(* Logix 5000 project; controller RN21_Architecture 1769-L16ER-BB1B rev 35.11; software revision 35.00; part 7 of 9 *)
(* tags used below, declared in another part *)
   ALMSrc_UniqueNum : DINT;
   AUDSrc : UDT_Audit;
   AUDSrc_UniqueNum : DINT;
   BMANSrc : UDT_Batch;
   BMANSrc_UniqueNum : DINT;
   FC_BMAN_Arch : AOI_BMAN_Arch;
   FC_TBC : AOI_TBC;
   FCI_AUDDataLogTrig : BOOL;
   FCI_BMANDataLogTrig : BOOL;
   HMI_CONTROL_SCREEN : DINT;
   HmiCurrentScreen : DINT;
   HMIOLDSCREENVALUE : DINT;
   HMISCREEN : BOOL;
   HMISCREENCHANGED : BOOL;
   inactivity_in_minutes : DINT;
   inactivity_time : DINT;
   INTERNAL_RN21_HB_PLC2ServerCommFailed : BOOL;
   INTERNAL_RN21_PLC2HMICommFailed : BOOL;
   LBSrc_UniqueNum : DINT;
   LoginDNDel : TIMER;
   PDLSrc_PDL_UID : DINT;
   PLC_HMI_CommTag : BOOL;
   PLC_RTC : DINT[7];
   Remaining_time : DINT;
   remaining_time_compareTag : DINT;
   RN21_AUD_BAMTrig : DINT[5];
   RN21_AUD_BAT_NTrig : DINT[4];
   RN21_AUD_BAT_PTrig : DINT[4];
   RN21_AUD_NETrig : DINT[11];
   RN21_AUDBAM_ONS : BOOL[128];
   RN21_AutoLogedOut : BOOL;
   RN21_BACK_BatchDataStatus : BOOL;   // BATCH START ACKNOWLEDGEMENT STATUS FROM SERVER
   RN21_BACK_BatchStartHMI : BOOL;   // HMI BATCH START IN BATCH DETAILS
   RN21_BACKONS : DINT[1];
   RN21_BMAN_BatchStarted : BOOL;   // BATCH STARTED IN BATCH MANAGEMENT
   RN21_BMAN_BatchStopped : BOOL;   // BATCH STOPPED IN BATCH MANAGEMENT
   RN21_BMAN_HMIBatchStart : BOOL;   // BATCH START
   RN21_BMAN_HMIBatchStop : BOOL;
   RN21_BMANBASTPNEG : BOOL;
   RN21_BMANBASTPPOS : BOOL;
   RN21_BMANBASTRTNEG : BOOL;
   RN21_BMANBASTRTPOS : BOOL;
   RN21_HB_PLC2ServerCommFailed : BOOL;
   RN21_LBStatus : INT;   // Login Block Status
   RN21_Map_BAM : BOOL[128];
   RN21_PLC2HMICommFailed : BOOL;
   RN21_RM_HMICODE : STRING;
   RN21_UMLogoutTag : INT;
   RPSrc_RP_UID : DINT;
   RTC_DATE_AND_TIME_UNLATCH_DELAY1 : TIMER;
   TMR_AutoLogout : TIMER;
   TMR_AutoLogoutRstDly : TIMER;
   TMR_BatchStartAckDlyRst : TIMER;
   TMR_BatchStrtdDlyStsMov : TIMER;
   TMR_HBSetDelay : TIMER;
   TMR_LogoutTagRst : TIMER;
   TMR_PHSetDelay : TIMER;
   TMR_PLCtoHMICommCheck : TIMER;
   TMR_PLCToSrvComCheck : TIMER;
   ALM_TriggerId : BOOL;
   ALM_UniqueNum : DINT;
   AUD_TriggerId : BOOL;
   AUD_UniqueNum : DINT;
   BACK_BATCH_NO : STRING;
   BACK_BatchStartACK : DINT;
   BACK_LOT_NO : STRING;
   BMAN_BatchUniqueId : DINT;
   BMAN_TriggerBit : BOOL;
   BMANSer : UDT_Batch;
   HB_HEART_BEAT : BOOL;
   LOGIN_TriggerId : BOOL;
   LOGIN_UniqueNum : DINT;
   PDL_Trigger : BOOL;
   PDL_UID : DINT;
   RN21_BACK_BatchSize : REAL;
   RN21_BACK_ProductCode : STRING;
   RN21_BACK_ProductName : STRING;
   RP_Trigger : BOOL;
   RP_UID : DINT;
   RTC_DAY : DINT;
   RTC_HOUR : DINT;
   RTC_MINUTE : DINT;
   RTC_MONTH : DINT;
   RTC_SAVE_DATE_AND_TIME : BOOL;
   RTC_SECONDS : DINT;
   RTC_UniqueId : DINT;
   RTC_YEAR : DINT;
   ServerRTC : DINT[8];
   TBC_ALARMBLOCK_PLCUID : DINT;
   TBC_ALARMBLOCK_SERVERUID : DINT;
   TBC_ALARMBLOCK_TRIGGER : BOOL;
   TBC_AUDITBLOCK_PLCUID : DINT;
   TBC_AUDITBLOCK_SERVERUID : DINT;
   TBC_AUDITBLOCK_TRIGGER : BOOL;
   TBC_BATCHMGMTBLOCK_PLCUID : DINT;
   TBC_BATCHMGMTBLOCK_SERVERUID : DINT;
   TBC_BATCHMGMTBLOCK_TRIGGER : BOOL;
   TBC_POSITION : DINT;
   TBC_PROCESSBLOCK_PLCUID : DINT;
   TBC_PROCESSBLOCK_SERVERUID : DINT;
   TBC_PROCESSBLOCK_TRIGGER : BOOL;
   TBC_RECIPEBLOCK_PLCUID : DINT;
   TBC_RECIPEBLOCK_SERVERUID : DINT;
   TBC_RECIPEBLOCK_TRIGGER : BOOL;
   TBC_UID : DINT;
   TBC_UMBLOCK_PLCUID : DINT;
   TBC_UMBLOCK_SERVERUID : DINT;
   TBC_UMBLOCK_TRIGGER : BOOL;
(* MainProgram, continued *)

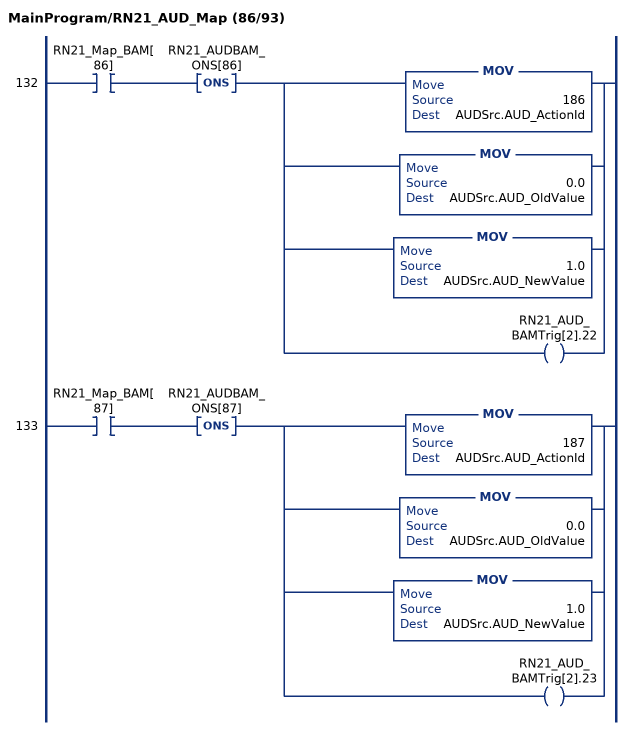
   [picture p168: MainProgram/RN21_AUD_Map rungs 132-133]
   132: XIC(RN21_Map_BAM[86])ONS(RN21_AUDBAM_ONS[86])[MOV(186,AUDSrc.AUD_ActionId) ,MOV(0.0,AUDSrc.AUD_OldValue) ,MOV(1.0,AUDSrc.AUD_NewValue) ,OTE(RN21_AUD_BAMTrig[2].22) ];
   133: XIC(RN21_Map_BAM[87])ONS(RN21_AUDBAM_ONS[87])[MOV(187,AUDSrc.AUD_ActionId) ,MOV(0.0,AUDSrc.AUD_OldValue) ,MOV(1.0,AUDSrc.AUD_NewValue) ,OTE(RN21_AUD_BAMTrig[2].23) ];
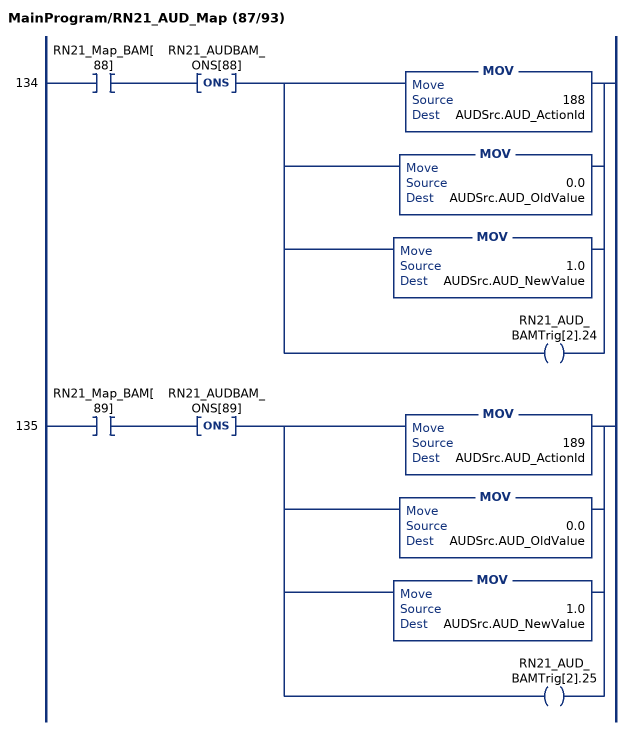
   134: XIC(RN21_Map_BAM[88])ONS(RN21_AUDBAM_ONS[88])[MOV(188,AUDSrc.AUD_ActionId) ,MOV(0.0,AUDSrc.AUD_OldValue) ,MOV(1.0,AUDSrc.AUD_NewValue) ,OTE(RN21_AUD_BAMTrig[2].24) ];
   135: XIC(RN21_Map_BAM[89])ONS(RN21_AUDBAM_ONS[89])[MOV(189,AUDSrc.AUD_ActionId) ,MOV(0.0,AUDSrc.AUD_OldValue) ,MOV(1.0,AUDSrc.AUD_NewValue) ,OTE(RN21_AUD_BAMTrig[2].25) ];
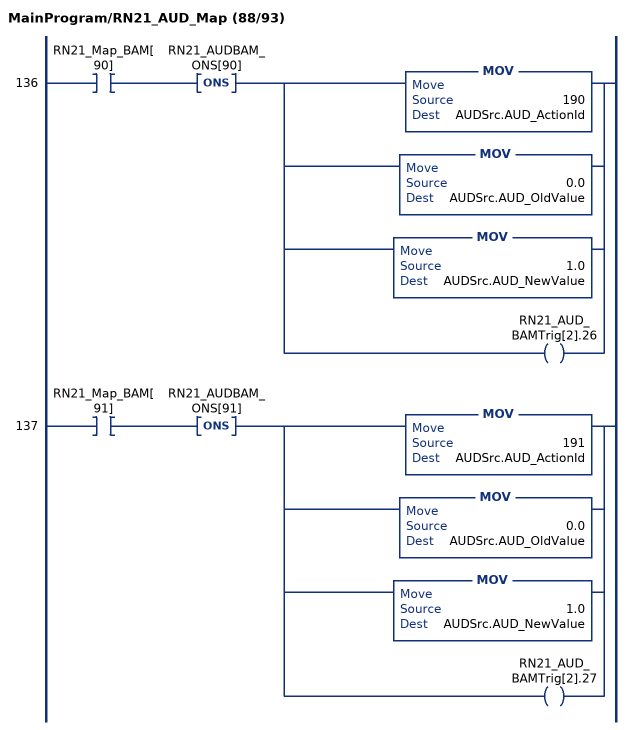
   136: XIC(RN21_Map_BAM[90])ONS(RN21_AUDBAM_ONS[90])[MOV(190,AUDSrc.AUD_ActionId) ,MOV(0.0,AUDSrc.AUD_OldValue) ,MOV(1.0,AUDSrc.AUD_NewValue) ,OTE(RN21_AUD_BAMTrig[2].26) ];
   137: XIC(RN21_Map_BAM[91])ONS(RN21_AUDBAM_ONS[91])[MOV(191,AUDSrc.AUD_ActionId) ,MOV(0.0,AUDSrc.AUD_OldValue) ,MOV(1.0,AUDSrc.AUD_NewValue) ,OTE(RN21_AUD_BAMTrig[2].27) ];
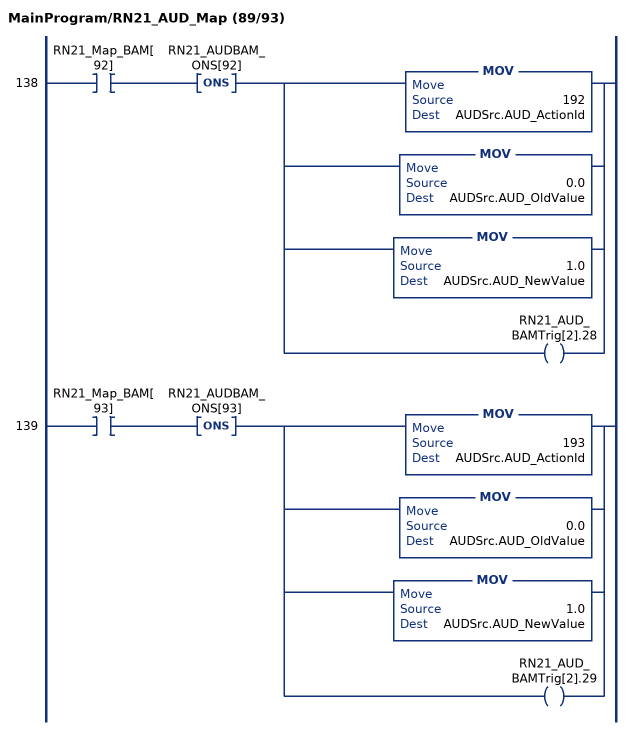
   138: XIC(RN21_Map_BAM[92])ONS(RN21_AUDBAM_ONS[92])[MOV(192,AUDSrc.AUD_ActionId) ,MOV(0.0,AUDSrc.AUD_OldValue) ,MOV(1.0,AUDSrc.AUD_NewValue) ,OTE(RN21_AUD_BAMTrig[2].28) ];
   139: XIC(RN21_Map_BAM[93])ONS(RN21_AUDBAM_ONS[93])[MOV(193,AUDSrc.AUD_ActionId) ,MOV(0.0,AUDSrc.AUD_OldValue) ,MOV(1.0,AUDSrc.AUD_NewValue) ,OTE(RN21_AUD_BAMTrig[2].29) ];
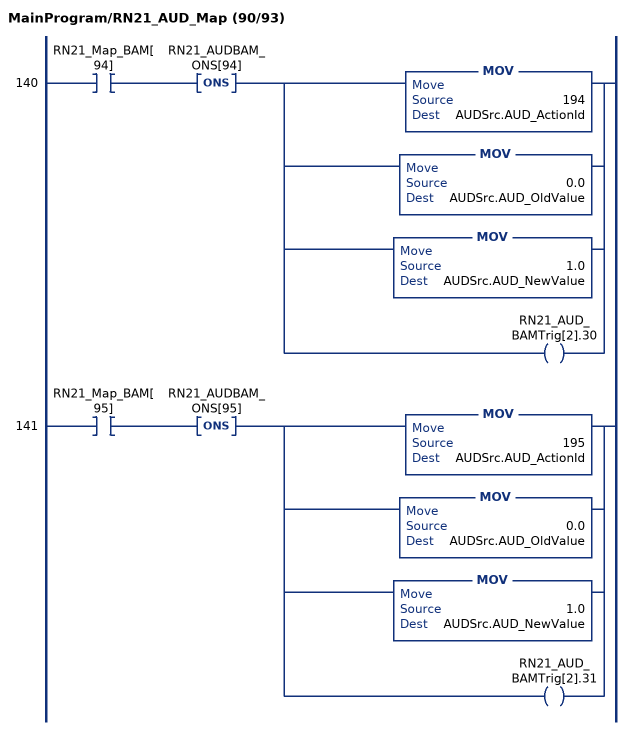
   140: XIC(RN21_Map_BAM[94])ONS(RN21_AUDBAM_ONS[94])[MOV(194,AUDSrc.AUD_ActionId) ,MOV(0.0,AUDSrc.AUD_OldValue) ,MOV(1.0,AUDSrc.AUD_NewValue) ,OTE(RN21_AUD_BAMTrig[2].30) ];
   141: XIC(RN21_Map_BAM[95])ONS(RN21_AUDBAM_ONS[95])[MOV(195,AUDSrc.AUD_ActionId) ,MOV(0.0,AUDSrc.AUD_OldValue) ,MOV(1.0,AUDSrc.AUD_NewValue) ,OTE(RN21_AUD_BAMTrig[2].31) ];
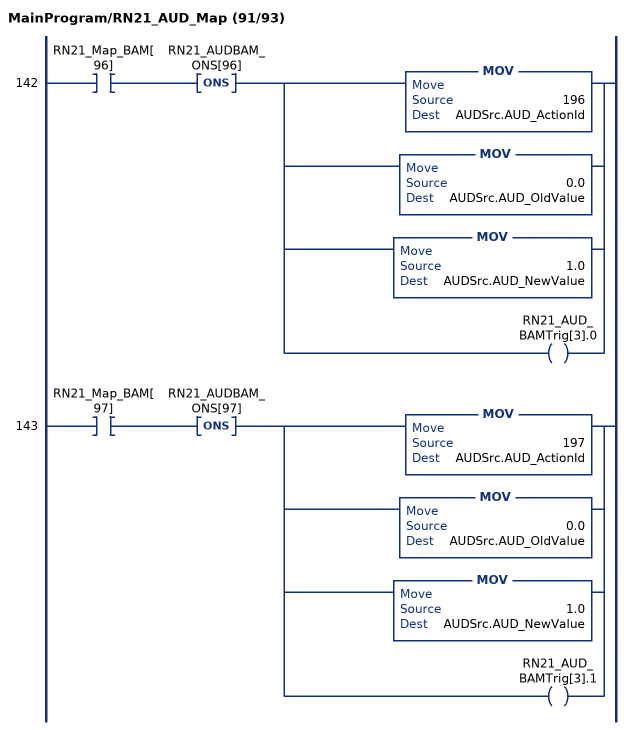
   142: XIC(RN21_Map_BAM[96])ONS(RN21_AUDBAM_ONS[96])[MOV(196,AUDSrc.AUD_ActionId) ,MOV(0.0,AUDSrc.AUD_OldValue) ,MOV(1.0,AUDSrc.AUD_NewValue) ,OTE(RN21_AUD_BAMTrig[3].0) ];
   143: XIC(RN21_Map_BAM[97])ONS(RN21_AUDBAM_ONS[97])[MOV(197,AUDSrc.AUD_ActionId) ,MOV(0.0,AUDSrc.AUD_OldValue) ,MOV(1.0,AUDSrc.AUD_NewValue) ,OTE(RN21_AUD_BAMTrig[3].1) ];
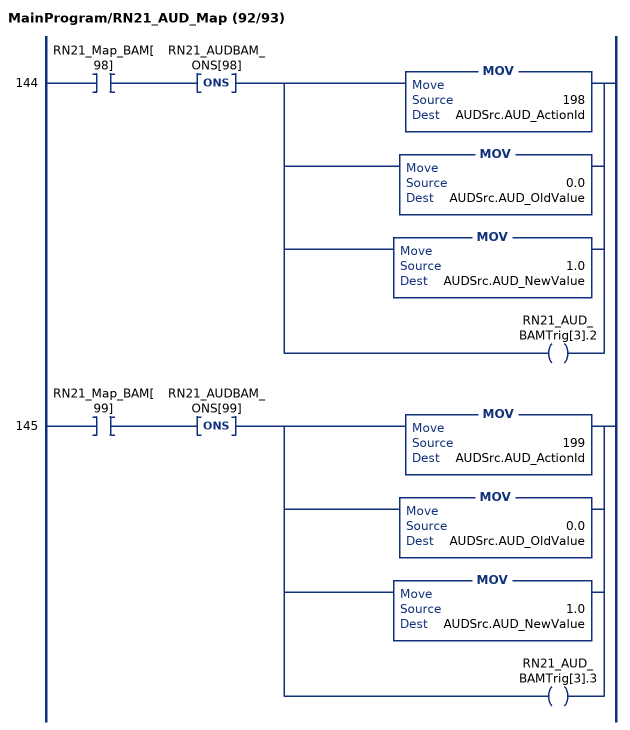
   144: XIC(RN21_Map_BAM[98])ONS(RN21_AUDBAM_ONS[98])[MOV(198,AUDSrc.AUD_ActionId) ,MOV(0.0,AUDSrc.AUD_OldValue) ,MOV(1.0,AUDSrc.AUD_NewValue) ,OTE(RN21_AUD_BAMTrig[3].2) ];
   145: XIC(RN21_Map_BAM[99])ONS(RN21_AUDBAM_ONS[99])[MOV(199,AUDSrc.AUD_ActionId) ,MOV(0.0,AUDSrc.AUD_OldValue) ,MOV(1.0,AUDSrc.AUD_NewValue) ,OTE(RN21_AUD_BAMTrig[3].3) ];
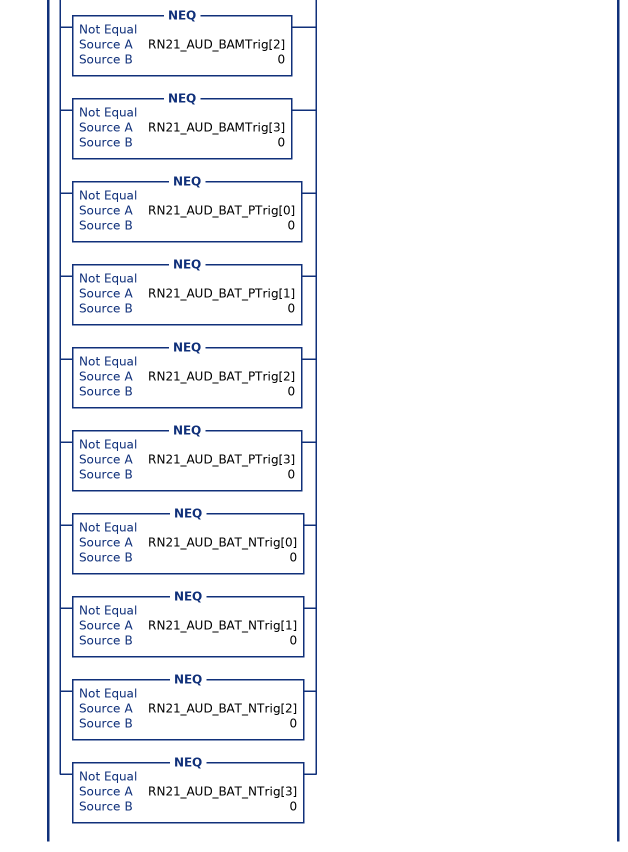
   146: [NEQ(RN21_AUD_NETrig[0],0) ,NEQ(RN21_AUD_NETrig[1],0) ,NEQ(RN21_AUD_NETrig[2],0) ,NEQ(RN21_AUD_NETrig[3],0) ,NEQ(RN21_AUD_NETrig[4],0) ,NEQ(RN21_AUD_NETrig[5],0) ,NEQ(RN21_AUD_NETrig[6],0) ,NEQ(RN21_AUD_NETrig[7],0) ,NEQ(RN21_AUD_NETrig[8],0) ,NEQ(RN21_AUD_NETrig[9],0) ,NEQ(RN21_AUD_BAMTrig[0],0) ,NEQ(RN21_AUD_BAMTrig[1],0) ,NEQ(RN21_AUD_BAMTrig[2],0) ,NEQ(RN21_AUD_BAMTrig[3],0) ,NEQ(RN21_AUD_BAT_PTrig[0],0) ,NEQ(RN21_AUD_BAT_PTrig[1],0) ,NEQ(RN21_AUD_BAT_PTrig[2],0) ,NEQ(RN21_AUD_BAT_PTrig[3],0) ,NEQ(RN21_AUD_BAT_NTrig[0],0) ,NEQ(RN21_AUD_BAT_NTrig[1],0) ,NEQ(RN21_AUD_BAT_NTrig[2],0) ,NEQ(RN21_AUD_BAT_NTrig[3],0) ]OTE(FCI_AUDDataLogTrig);
END_ROUTINE

ROUTINE RN21_BMAN_Main   (* ladder *)
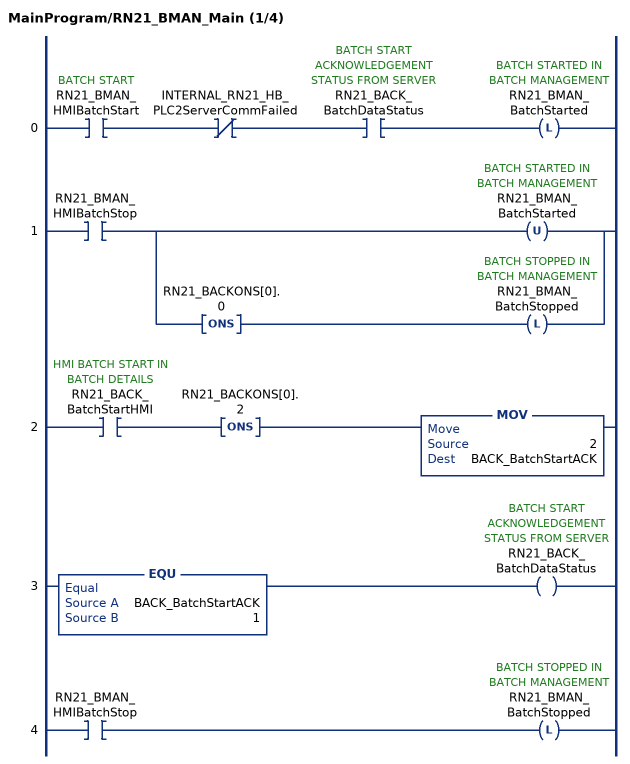
   0: XIC(RN21_BMAN_HMIBatchStart)XIO(INTERNAL_RN21_HB_PLC2ServerCommFailed)XIC(RN21_BACK_BatchDataStatus)OTL(RN21_BMAN_BatchStarted);
   1: XIC(RN21_BMAN_HMIBatchStop)[OTU(RN21_BMAN_BatchStarted) ,ONS(RN21_BACKONS[0].0) OTL(RN21_BMAN_BatchStopped) ];
   2: XIC(RN21_BACK_BatchStartHMI)ONS(RN21_BACKONS[0].2)MOV(2,BACK_BatchStartACK);
   3: EQU(BACK_BatchStartACK,1)OTE(RN21_BACK_BatchDataStatus);
   4: XIC(RN21_BMAN_HMIBatchStop)OTL(RN21_BMAN_BatchStopped);
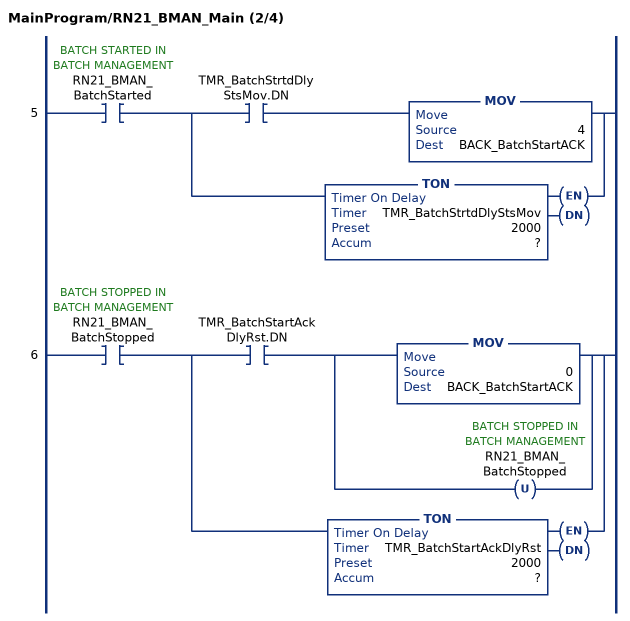
   5: XIC(RN21_BMAN_BatchStarted)[XIC(TMR_BatchStrtdDlyStsMov.DN) MOV(4,BACK_BatchStartACK) ,TON(TMR_BatchStrtdDlyStsMov,?,?) ];
   6: XIC(RN21_BMAN_BatchStopped)[XIC(TMR_BatchStartAckDlyRst.DN) [MOV(0,BACK_BatchStartACK) ,OTU(RN21_BMAN_BatchStopped) ] ,TON(TMR_BatchStartAckDlyRst,?,?) ];
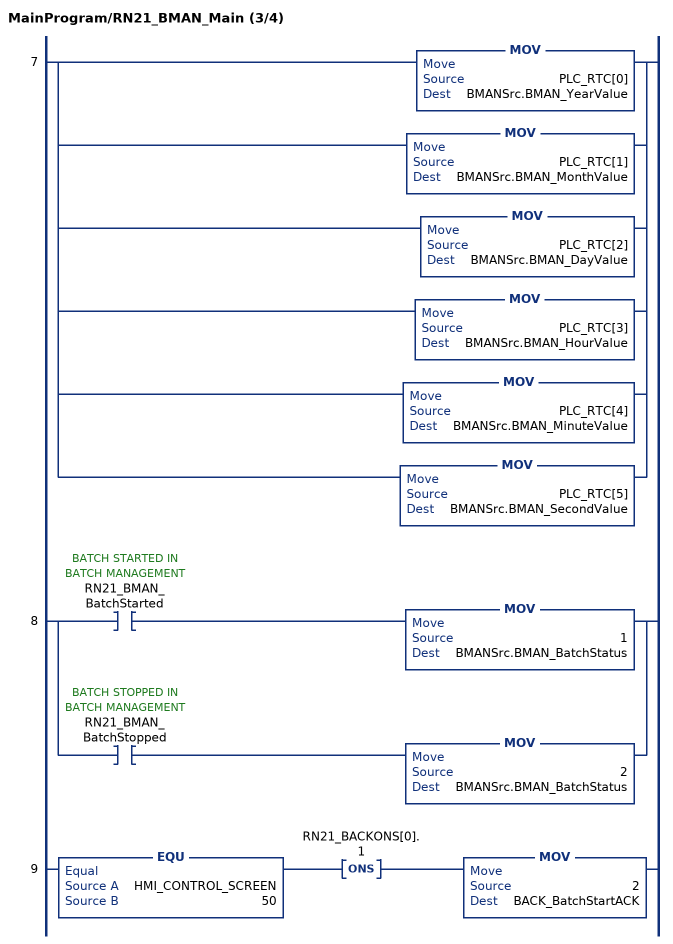
   7: [MOV(PLC_RTC[0],BMANSrc.BMAN_YearValue) ,MOV(PLC_RTC[1],BMANSrc.BMAN_MonthValue) ,MOV(PLC_RTC[2],BMANSrc.BMAN_DayValue) ,MOV(PLC_RTC[3],BMANSrc.BMAN_HourValue) ,MOV(PLC_RTC[4],BMANSrc.BMAN_MinuteValue) ,MOV(PLC_RTC[5],BMANSrc.BMAN_SecondValue) ];
   8: [XIC(RN21_BMAN_BatchStarted) MOV(1,BMANSrc.BMAN_BatchStatus) ,XIC(RN21_BMAN_BatchStopped) MOV(2,BMANSrc.BMAN_BatchStatus) ];
   9: EQU(HMI_CONTROL_SCREEN,50)ONS(RN21_BACKONS[0].1)MOV(2,BACK_BatchStartACK);
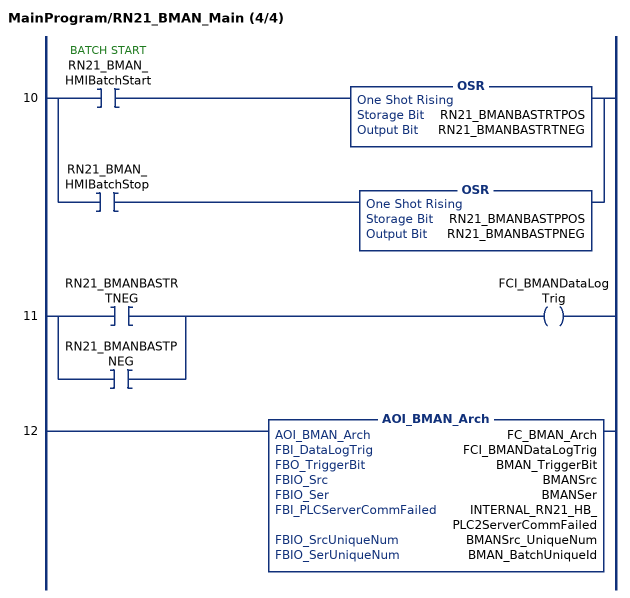
   10: [XIC(RN21_BMAN_HMIBatchStart) OSR(RN21_BMANBASTRTPOS,RN21_BMANBASTRTNEG) ,XIC(RN21_BMAN_HMIBatchStop) OSR(RN21_BMANBASTPPOS,RN21_BMANBASTPNEG) ];
   11: [XIC(RN21_BMANBASTRTNEG) ,XIC(RN21_BMANBASTPNEG) ]OTE(FCI_BMANDataLogTrig);
   12: AOI_BMAN_Arch(FC_BMAN_Arch,FCI_BMANDataLogTrig,BMAN_TriggerBit,BMANSrc,BMANSer,INTERNAL_RN21_HB_PLC2ServerCommFailed,BMANSrc_UniqueNum,BMAN_BatchUniqueId);
END_ROUTINE

ROUTINE RN21_BMAN_Map   (* ladder *)
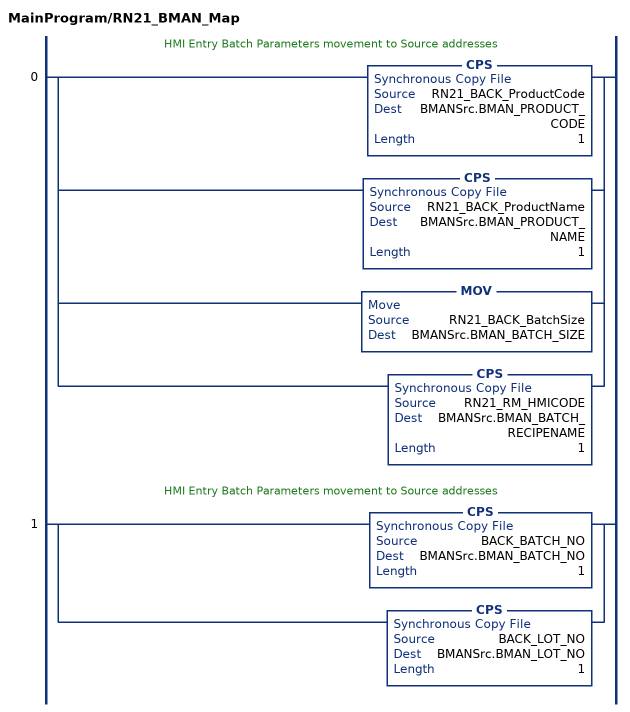
   // HMI Entry Batch Parameters movement to Source addresses
   0: [CPS(RN21_BACK_ProductCode,BMANSrc.BMAN_PRODUCT_CODE,1) ,CPS(RN21_BACK_ProductName,BMANSrc.BMAN_PRODUCT_NAME,1) ,MOV(RN21_BACK_BatchSize,BMANSrc.BMAN_BATCH_SIZE) ,CPS(RN21_RM_HMICODE,BMANSrc.BMAN_BATCH_RECIPENAME,1) ];
   // HMI Entry Batch Parameters movement to Source addresses
   1: [CPS(BACK_BATCH_NO,BMANSrc.BMAN_BATCH_NO,1) ,CPS(BACK_LOT_NO,BMANSrc.BMAN_LOT_NO,1) ];
END_ROUTINE

ROUTINE RN21_Global   (* ladder *)
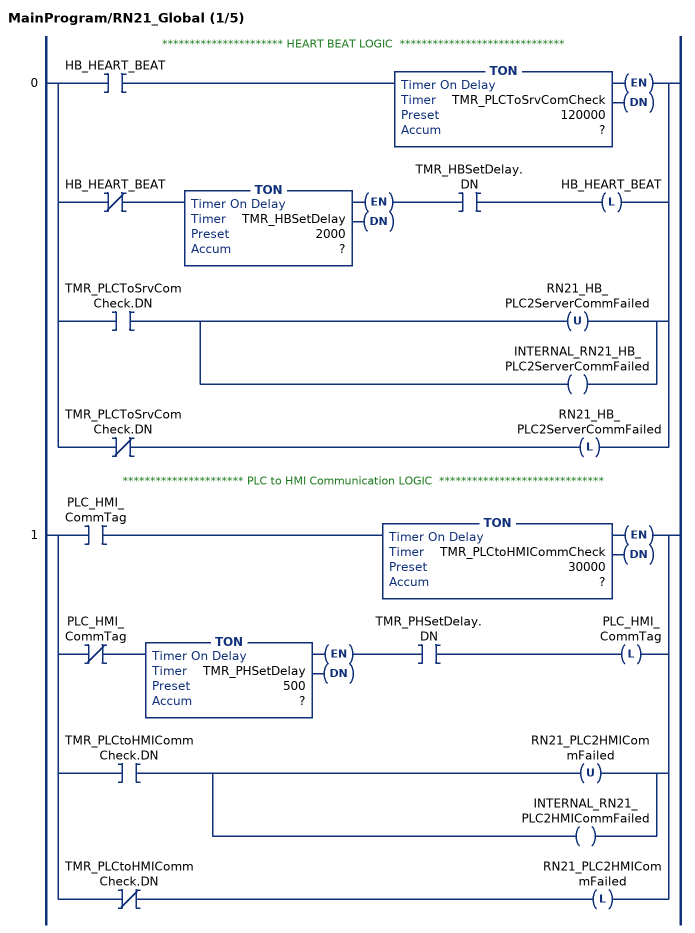
   // ********************** HEART BEAT LOGIC  ******************************
   0: [XIC(HB_HEART_BEAT) TON(TMR_PLCToSrvComCheck,?,?) ,XIO(HB_HEART_BEAT) TON(TMR_HBSetDelay,?,?) XIC(TMR_HBSetDelay.DN) OTL(HB_HEART_BEAT) ,XIC(TMR_PLCToSrvComCheck.DN) [OTU(RN21_HB_PLC2ServerCommFailed) ,OTE(INTERNAL_RN21_HB_PLC2ServerCommFailed) ] ,XIO(TMR_PLCToSrvComCheck.DN) OTL(RN21_HB_PLC2ServerCommFailed) ];
   // ********************** PLC to HMI Communication LOGIC  ******************************
   1: [XIC(PLC_HMI_CommTag) TON(TMR_PLCtoHMICommCheck,?,?) ,XIO(PLC_HMI_CommTag) TON(TMR_PHSetDelay,?,?) XIC(TMR_PHSetDelay.DN) OTL(PLC_HMI_CommTag) ,XIC(TMR_PLCtoHMICommCheck.DN) [OTU(RN21_PLC2HMICommFailed) ,OTE(INTERNAL_RN21_PLC2HMICommFailed) ] ,XIO(TMR_PLCtoHMICommCheck.DN) OTL(RN21_PLC2HMICommFailed) ];
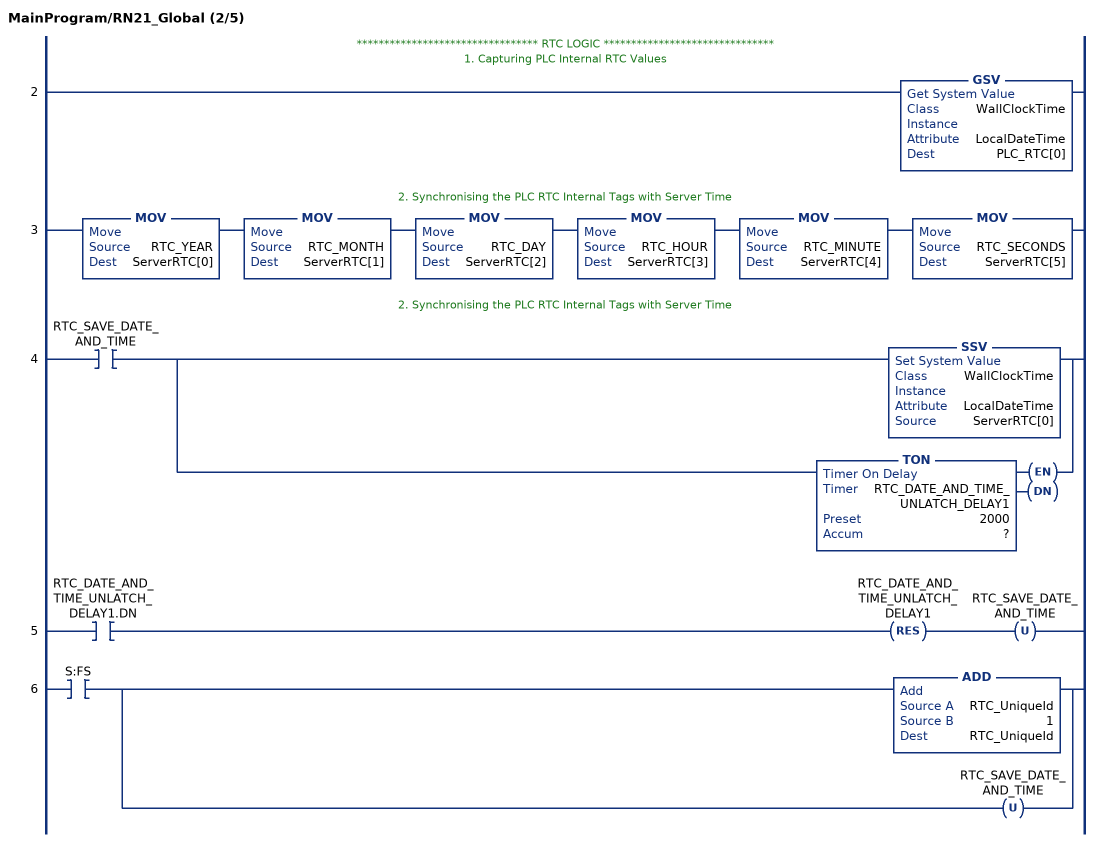
   // ********************************* RTC LOGIC *******************************
   // 1. Capturing PLC Internal RTC Values
   2: GSV(WallClockTime,,LocalDateTime,PLC_RTC[0]);
   // 2. Synchronising the PLC RTC Internal Tags with Server Time
   3: MOV(RTC_YEAR,ServerRTC[0])MOV(RTC_MONTH,ServerRTC[1])MOV(RTC_DAY,ServerRTC[2])MOV(RTC_HOUR,ServerRTC[3])MOV(RTC_MINUTE,ServerRTC[4])MOV(RTC_SECONDS,ServerRTC[5]);
   // 2. Synchronising the PLC RTC Internal Tags with Server Time
   4: XIC(RTC_SAVE_DATE_AND_TIME)[SSV(WallClockTime,,LocalDateTime,ServerRTC[0]) ,TON(RTC_DATE_AND_TIME_UNLATCH_DELAY1,?,?) ];
   5: XIC(RTC_DATE_AND_TIME_UNLATCH_DELAY1.DN)RES(RTC_DATE_AND_TIME_UNLATCH_DELAY1)OTU(RTC_SAVE_DATE_AND_TIME);
   6: XIC(S:FS)[ADD(RTC_UniqueId,1,RTC_UniqueId) ,OTU(RTC_SAVE_DATE_AND_TIME) ];
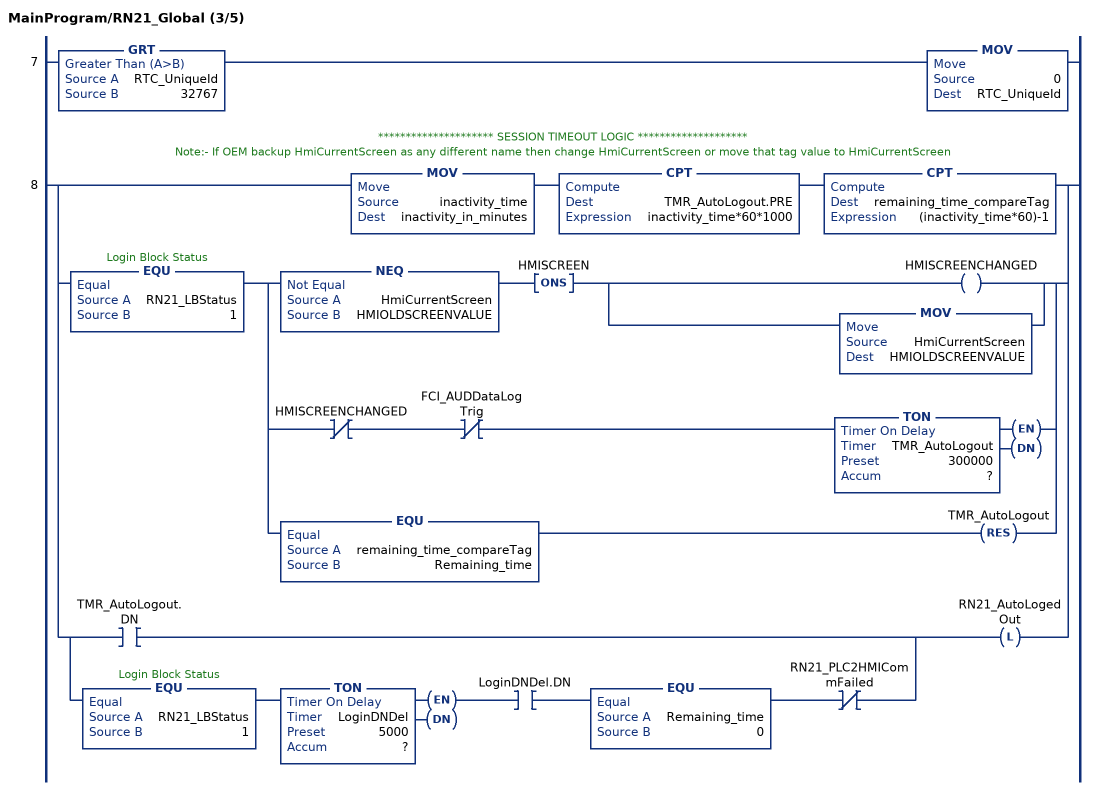
   7: GRT(RTC_UniqueId,32767)MOV(0,RTC_UniqueId);
   // ********************* SESSION TIMEOUT LOGIC ********************
   // Note:- If OEM backup HmiCurrentScreen as any different name then change HmiCurrentScreen or move that tag value to HmiCurrentScreen
   8: [MOV(inactivity_time,inactivity_in_minutes) CPT(TMR_AutoLogout.PRE,inactivity_time*60*1000) CPT(remaining_time_compareTag,(inactivity_time*60)-1) ,EQU(RN21_LBStatus,1) [NEQ(HmiCurrentScreen,HMIOLDSCREENVALUE) ONS(HMISCREEN) [OTE(HMISCREENCHANGED) ,MOV(HmiCurrentScreen,HMIOLDSCREENVALUE) ] ,XIO(HMISCREENCHANGED) XIO(FCI_AUDDataLogTrig) TON(TMR_AutoLogout,?,?) ,EQU(remaining_time_compareTag,Remaining_time) RES(TMR_AutoLogout) ] ,[XIC(TMR_AutoLogout.DN) ,EQU(RN21_LBStatus,1) TON(LoginDNDel,?,?) XIC(LoginDNDel.DN) EQU(Remaining_time,0) XIO(RN21_PLC2HMICommFailed) ] OTL(RN21_AutoLogedOut) ];
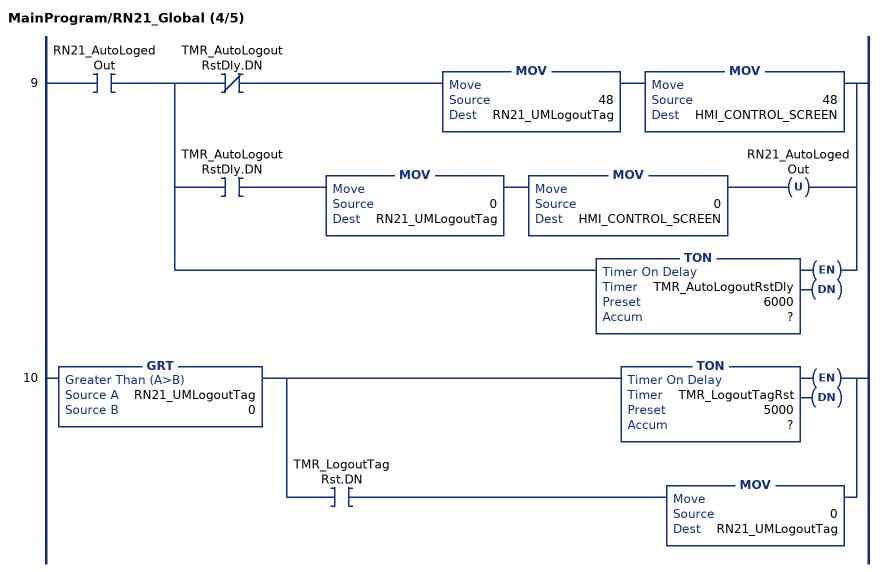
   9: XIC(RN21_AutoLogedOut)[XIO(TMR_AutoLogoutRstDly.DN) MOV(48,RN21_UMLogoutTag) MOV(48,HMI_CONTROL_SCREEN) ,XIC(TMR_AutoLogoutRstDly.DN) MOV(0,RN21_UMLogoutTag) MOV(0,HMI_CONTROL_SCREEN) OTU(RN21_AutoLogedOut) ,TON(TMR_AutoLogoutRstDly,?,?) ];
   10: GRT(RN21_UMLogoutTag,0)[TON(TMR_LogoutTagRst,?,?) ,XIC(TMR_LogoutTagRst.DN) MOV(0,RN21_UMLogoutTag) ];
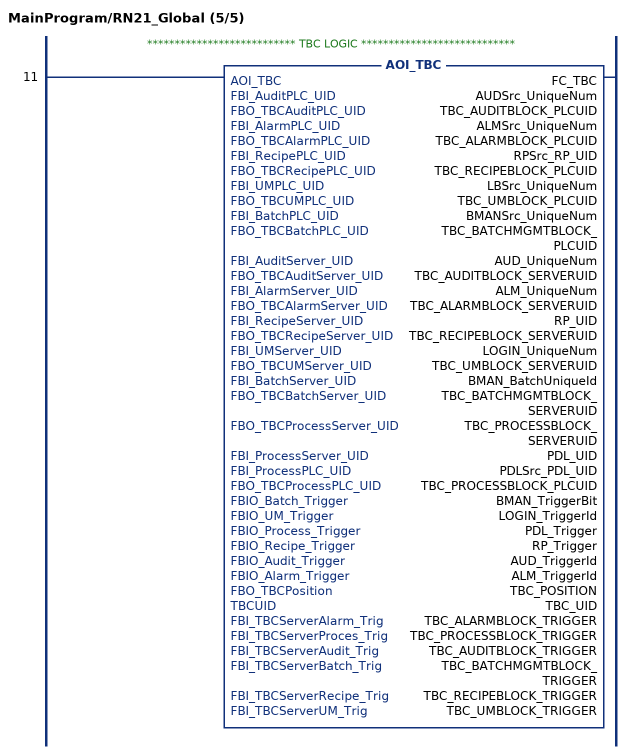
   // *************************** TBC LOGIC ****************************
   11: AOI_TBC(FC_TBC,AUDSrc_UniqueNum,TBC_AUDITBLOCK_PLCUID,ALMSrc_UniqueNum,TBC_ALARMBLOCK_PLCUID,RPSrc_RP_UID,TBC_RECIPEBLOCK_PLCUID,LBSrc_UniqueNum,TBC_UMBLOCK_PLCUID,BMANSrc_UniqueNum,TBC_BATCHMGMTBLOCK_PLCUID,AUD_UniqueNum,TBC_AUDITBLOCK_SERVERUID,ALM_UniqueNum,TBC_ALARMBLOCK_SERVERUID,RP_UID,TBC_RECIPEBLOCK_SERVERUID,LOGIN_UniqueNum,TBC_UMBLOCK_SERVERUID,BMAN_BatchUniqueId,TBC_BATCHMGMTBLOCK_SERVERUID,TBC_PROCESSBLOCK_SERVERUID,PDL_UID,PDLSrc_PDL_UID,TBC_PROCESSBLOCK_PLCUID,BMAN_TriggerBit,LOGIN_TriggerId,PDL_Trigger,RP_Trigger,AUD_TriggerId,ALM_TriggerId,TBC_POSITION,TBC_UID,TBC_ALARMBLOCK_TRIGGER,TBC_PROCESSBLOCK_TRIGGER,TBC_AUDITBLOCK_TRIGGER,TBC_BATCHMGMTBLOCK_TRIGGER,TBC_RECIPEBLOCK_TRIGGER,TBC_UMBLOCK_TRIGGER);
END_ROUTINE
